TYPE ST_ClockDefaultParameters :
STRUCT
	tTaskCycleTime : TIME := GlobalVariables.tCtrlCycleTime_MAIN;
	tCtrlCycleTime : TIME := GlobalVariables.tCtrlCycleTime_MAIN;
END_STRUCT
END_TYPE

(* stored: Version 1.1.0.1, ProductVersion 3.1.4024.10
   DUT ST_ClockDefaultParameters: Id {e67b2ea3-fe26-46dd-9e02-fb491d9b8c40} *)
